FUNCTION TFPalletizerPackValidation : INT
VAR_INPUT
	WorkArea : POINTER TO ARRAY [1..MAXAREA] OF TFMachinePalletizer_WorkArea;
	WorkAreaState : POINTER TO ARRAY [1..MAXAREA] OF TFMachinePalletizer_WorkAreaState;
	WorkPickPointState : POINTER TO ARRAY [1..MAXPICKPOINT] OF TFMachinePalletizer_WorkPickPointState;
	Forming : POINTER TO ARRAY [1..MAXFORMING] OF TFMachinePalletizer_Forming;
	Mission : POINTER TO TFMachinePalletizer_Mission;
	AxisPar : POINTER TO Ax_Palletizer_Parameters;
END_VAR
VAR
	wpp : INT;
	i : INT;
	PackOffset : REAL;
	CodeAssignedToWA : BOOL; // TRUE se i codice è assegnato ad almeno una WA
	fcode : INT;
END_VAR

TFPalletizerPackValidation := 0; 
PackOffset := 50.0;

IF  Mission^.KPick >= AxisPar^.MaxPosition OR Mission^.KPick <= AxisPar^.MinPosition// OR
	(*Mission^.KPlace > AxisPar^.K.MaxPosition OR Mission^.KPlace < AxisPar^.K.MinPosition*) THEN
		TFPalletizerPackValidation := ErrCONFIGURAZIONEPINZASABGLIATA; // Configurazione Pinza non adatta al prelievo o al deposito
		RETURN;	
END_IF

FOR wpp:=1 TO MAXPICKPOINT DO
	(* Verifico disponibilità Pacco *)
	IF WorkPickPointState^[wpp].State = WORKPICKPOINT_PRODOTTO_PRESENTE THEN
		fcode := TFPalletizerGetFormingFromCode(Forming,WorkPickPointState^[wpp].Code);
		CASE TIPO_RIBALTINO OF
			RIBALTINO_DOPO_SQUADRO:
				IF fcode = 0 THEN
					TFPalletizerPackValidation := ErrPACKCODENOTVALID; // Codice non associato a formatura
					RETURN;			
				ELSIF (WorkPickPointState^[wpp].XDim < Forming^[fcode].PX - PackOffset OR
					WorkPickPointState^[wpp].XDim > Forming^[fcode].PX + PackOffset) OR
					(WorkPickPointState^[wpp].YDim < Forming^[fcode].PY - PackOffset  OR
					WorkPickPointState^[wpp].YDim > Forming^[fcode].PY + PackOffset) OR
					(WorkPickPointState^[wpp].ZDim < Forming^[fcode].PZ - PackOffset OR
					WorkPickPointState^[wpp].ZDim > Forming^[fcode].PZ + PackOffset)THEN
						TFPalletizerPackValidation := ErrPACKDIMENSIONNOTVALID; // Grandezze pacco errate
						RETURN;
				END_IF

			RIBALTINO_DIRETTO:
				IF fcode = 0 THEN
					TFPalletizerPackValidation := ErrPACKCODENOTVALID; // Codice non associato a formatura
					RETURN;			
				ELSIF (WorkPickPointState^[wpp].XDim < Forming^[fcode].PY - PackOffset OR
					WorkPickPointState^[wpp].XDim > Forming^[fcode].PY + PackOffset) OR
					(WorkPickPointState^[wpp].YDim < Forming^[fcode].PX - PackOffset  OR
					WorkPickPointState^[wpp].YDim > Forming^[fcode].PX + PackOffset) OR
					(WorkPickPointState^[wpp].ZDim < Forming^[fcode].PZ - PackOffset OR
					WorkPickPointState^[wpp].ZDim > Forming^[fcode].PZ + PackOffset)THEN
						TFPalletizerPackValidation := ErrPACKDIMENSIONNOTVALID; // Grandezze pacco errate
						RETURN;
				END_IF	
		END_CASE
		
	END_IF
END_FOR	

(*FOR wpp:=1 TO MAXPICKPOINT DO
	(* Verifico disponibilità Pacco *)
	IF WorkPickPointState^[wpp].State = WORKPICKPOINT_PRODOTTO_PRESENTE THEN
		(* Verifico se il codice è assegnato a qualche workarea e se la formatura è attiva *)
		FOR i:=1 TO MAXAREA DO
			IF WorkPickPointState^[wpp].Code = WorkArea^[i].Code AND WorkArea^[i].Typology = TYPOLOGY_PALLET THEN
				//CodeAssignedToWA := TRUE;
				IF WorkArea^[i].Enable = 1 AND Forming^[WorkAreaState^[i].F].Enable = 0 THEN
					TFPalletizerPackValidation := 1;//codice assegnato a workarea con formatura disabilitata
					//RETURN;
				ELSIF  WorkArea^[i].Enable = 0 AND Forming^[WorkAreaState^[i].F].Enable = 1 THEN
					TFPalletizerPackValidation := 2;//codice assegnato a workarea disabilitata
					//RETURN;
				ELSIF WorkArea^[i].Enable = 0 AND  Forming^[WorkAreaState^[i].F].Enable = 0 THEN
					TFPalletizerPackValidation := 3;//codice assegnato a workarea disabilitata e con formatura disabilitata
					//RETURN;
				ELSE
					TFPalletizerPackValidation := 0;
					//RETURN;
				END_IF
			END_IF
		END_FOR	
	END_IF
	//TFPalletizerPackValidation := 4; // Codice pacco non assegnato a nessuna workarea
END_FOR
RETURN;*)
TFPalletizerPackValidation := 0;

END_FUNCTION

(* stored: Version 1.1.0.1, ProductVersion 3.1.4024.11
   POU TFPalletizerPackValidation: Id {766694d9-2ec8-4d75-ad9a-2c2aa2fc2e96}, SpecialFunc None *)
